TYPE TcoAbbRobotics_Status_v_1_x_x : STRUCT
    ActionDescription : STRING(100);
    State : TcoAbbRobotics_State_v_1_x_x;
END_STRUCT
END_TYPE

(* stored: Version 1.1.0.1, ProductVersion 3.1.4024.12
   DUT TcoAbbRobotics_Status_v_1_x_x: Id {3700e50f-c9cf-0135-026f-b0fcb141462e} *)
